(* PLC project op_shuttle, Dassault Systèmes ControlBuild 2024x *)
(* stored: creationDateTime 2023-10-03T11:13:59-01:00 *)

PROGRAM tri_chain.op_shuttle
  VAR_INPUT
    forward : BOOL := false;
    backward : BOOL := false;
    chainMotorOn : BOOL := false;
  END_VAR
  VAR_OUTPUT
    sensor_Pos1 : BOOL := false;
    sensor_Pos2 : BOOL := false;
    sensor_Pos3 : BOOL := false;
    end_sensor : BOOL := false;
  END_VAR

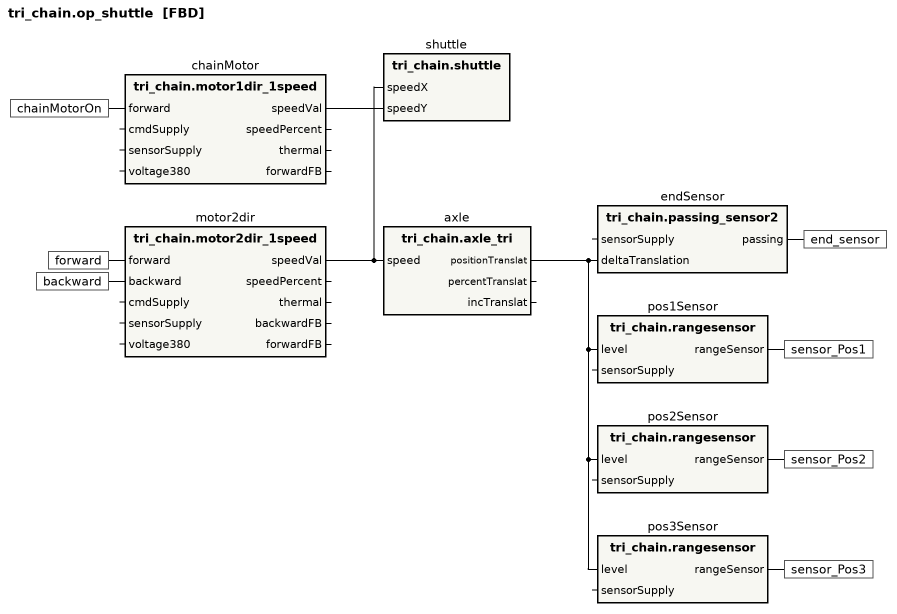
(* FBD diagram, written out as Structured Text *)
motor2dir(forward := forward, backward := backward);
axle(speed := motor2dir.speedVal);
pos1Sensor(level := axle.positionTranslat);
sensor_Pos1 := pos1Sensor.rangeSensor;
pos2Sensor(level := axle.positionTranslat);
sensor_Pos2 := pos2Sensor.rangeSensor;
pos3Sensor(level := axle.positionTranslat);
sensor_Pos3 := pos3Sensor.rangeSensor;
endSensor(deltaTranslation := axle.positionTranslat);
end_sensor := endSensor.passing;
chainMotor(forward := chainMotorOn);
shuttle(speedX := motor2dir.speedVal, speedY := chainMotor.speedVal);
END_PROGRAM
